{attribute 'GeneratedUsingTerminal: EL2564-0000-0016'}
{attribute addProperty BoxType "EL2564-0000-0016"}
{attribute addProperty Id "PWM_outputAT %Q*INT2"}
{attribute addProperty CRC "3606073277"}
{attribute addProperty Size "2"}
TYPE PWM_Outputs_Channel_D6F04FBD :
STRUCT
	{attribute addProperty Name "PWM_output"}
	PWM_output AT %Q* : INT;
END_STRUCT
END_TYPE

(* stored: Version 1.2.0.0, ProductVersion 3.1.4024.9
   DUT PWM_Outputs_Channel_D6F04FBD: Id {794f49b1-2da6-457f-a344-86718f04a7cf} *)
